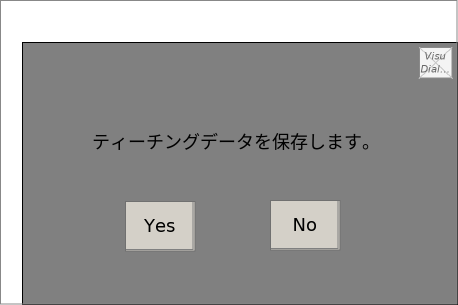
VISUALIZATION d_saveBtn  // 458x305
    Rectangle (22,42 436x263)
    Image (419,47 33x31), image: VisuDialogs.ImagePoolDialogs.Delete
        OnMouseClick: CloseDialog Dialog=d_saveBtn, Result=OK, NumpadKeypadSet=True
    Label (60,115 352x55), "ティーチングデータを保存します。"
    Button (125,201 70x50), "Yes"
        tap gvl_visu.flg_btn_savePalletize
        OnMouseClick: CloseDialog Dialog=d_saveBtn, Result=OK, NumpadKeypadSet=True
    Button (270,200 70x50), "No"
        OnMouseClick: CloseDialog Dialog=d_saveBtn, Result=OK, NumpadKeypadSet=True
END_VISUALIZATION

(* stored: Version 1.1.0.1, ProductVersion 3.1.4024.12
   Visu d_saveBtn: Id {2874b7f6-cf04-411d-aab0-e9eaaab96d25} *)
